TYPE ST_BHKW_Stellwert :
STRUCT
	Betrieb		: BOOL;
	Leistung		: USINT;
	Freigabe		: BOOL;
END_STRUCT
END_TYPE

(* stored: Version 1.1.0.1, ProductVersion 3.1.4024.9
   DUT ST_BHKW_Stellwert: Id {43220451-4e1f-41de-b244-3b94dae694c0} *)
